// TIA Portal V17 export
// export: Created 2023-12-05T13:40:24.3426745Z, ExportSetting WithDefaults, DisplayName Totally Integrated Automation Portal, DisplayVersion V17, DisplayName TIA Portal Openness, DisplayVersion V17, DisplayName TIA Portal Version Control Interface, DisplayVersion V17, DisplayName SINAMICS Startdrive Advanced, DisplayVersion V17, DisplayName SINAMICS Startdrive G130, G150, S120, S150, SINAMICS MV, S210, DisplayVersion V17, DisplayName SINAMICS Startdrive G110M, G120, G120C, G120D, G120P, G115D, DisplayVersion V17, DisplayName STEP 7 Professional, DisplayVersion V17, DisplayName STEP 7 Safety, DisplayVersion V17, DisplayName WinCC Professional, DisplayVersion V17
DATA_BLOCK "DB401 Counters machine"   // DB401
VERSION : 0.1
// stored: AutoNumber false, DBAccessibleFromOPCUA true, DBAccessibleFromWebserver true, InstanceOfName FB401 Counters machine, InstanceOfType FB
"FB401 Counters machine"
   // VAR_INPUT
   //    "ST2 Status" : Struct
   //       Good : Bool;
   //       Bad : Bool;
   //       Doubtful : Bool;
   //    END_STRUCT;
   //    "ST3 Status" : Struct
   //       Good : Bool;
   //       Bad : Bool;
   //       Doubtful : Bool;
   //    END_STRUCT;
   //    "ST4 Status" : Struct
   //       Good : Bool;
   //       Bad : Bool;
   //       Doubtful : Bool;
   //    END_STRUCT;
   //    "Unloading Status" : Struct
   //       Good : Bool;
   //       Bad : Bool;
   //       Doubtful : Bool;
   //    END_STRUCT;
   // END_VAR
   // VAR RETAIN
   //    Spare : Int;
   //    "Station 2" { S7_SetPoint := 'True'} : "FB400 Counters";
   //    "Station 3" { S7_SetPoint := 'True'} : "FB400 Counters";
   //    "Station 4" { S7_SetPoint := 'True'} : "FB400 Counters";
   //    "Station 1" { S7_SetPoint := 'True'} : "FB400 Counters";
   //    Names { S7_SetPoint := 'True'} : "VersionsNames";
   // END_VAR
BEGIN
END_DATA_BLOCK
